FUNCTION_BLOCK FB_ListString
VAR_INPUT
END_VAR
VAR_OUTPUT
END_VAR
VAR
	asList	: ARRAY[0..MAX_INDEX] OF STRING;
END_VAR
VAR CONSTANT
	MAX_INDEX	: INT := 9;
END_VAR


// FIFO

METHOD addEntry : BOOL
VAR_INPUT
	entry	: STRING;
END_VAR
VAR
	i	: INT;
END_VAR

addEntry := FALSE;
FOR i := 0 TO MAX_INDEX DO
	IF asList[i] = '' THEN
		asList[i] := entry;
		addEntry := TRUE;
		EXIT;
	END_IF
END_FOR
END_METHOD

METHOD PUBLIC clear : BOOL
VAR_INPUT
END_VAR
VAR
	i	: INT;
END_VAR

FOR i := 0 TO MAX_INDEX DO
	asList[i] := '';
END_FOR
END_METHOD

METHOD PUBLIC isEmpty : BOOL
VAR_INPUT
END_VAR

isEmpty := asList[0] = '';
END_METHOD

METHOD PUBLIC popEntry : STRING
VAR_INPUT
END_VAR
VAR
	i	: INT;
END_VAR

// return element
popEntry := asList[0];

// shift elements in array
FOR i := 0 TO MAX_INDEX - 1 DO
	asList[i] := asList[i + 1];
END_FOR
asList[MAX_INDEX] := '';
END_METHOD

END_FUNCTION_BLOCK

(* stored: Version 1.1.0.1, ProductVersion 3.1.4026.18
   POU FB_ListString: Id {bd4c7694-608d-4826-a99a-8bf4f1eb78cd}, SpecialFunc None
   Method addEntry: Id {91c1d7c7-509d-493d-80ac-3487cf502d84}
   Method clear: Id {9bfa52b7-5859-4429-b425-94fa111d7d90}
   Method isEmpty: Id {ac83f3d1-9d95-4cf6-b54a-8c5eb70f58fd}
   Method popEntry: Id {23c967e6-b739-4837-82a3-6c6b819d1543} *)
